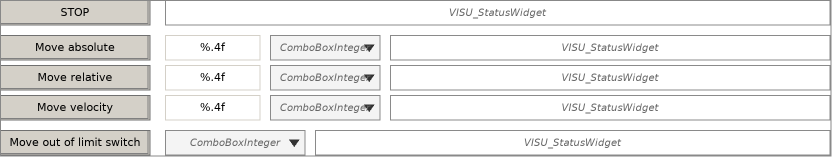
VISUALIZATION VISU_Axes_Commands_Movement  // 832x157
VAR_IN_OUT
    stop : AxesStopProcess;
    moveOutOfLimitSwitch : AxesMoveOutOfLimitSwitchProcess;
    moveAbsolute : AxesMoveAbsoluteProcess;
    moveRelative : AxesMoveRelativeProcess;
    moveVelocity : AxesMoveVelocityProcess;
    
    stopStatus : StatusWidget;
    moveOutOfLimitSwitchStatus : StatusWidget;
    moveAbsoluteStatus : StatusWidget;
    moveRelativeStatus : StatusWidget;
    moveVelocityStatus : StatusWidget;
END_VAR
    Button (0,0 150x25), "STOP", input disabled if: stop.statuses.enabledStatus.disabled
        OnMouseClick: execute { stop.request(); }
    Frame (165,0 665x25)
        shows VISU_StatusWidget(widget := stopStatus)
    Button (0,130 150x25), "Move out of limit switch", input disabled if: moveOutOfLimitSwitch.statuses.enabledStatus.disabled
        OnMouseClick: execute { moveOutOfLimitSwitch.do_request := TRUE; }
    Frame (315,130 515x25)
        shows VISU_StatusWidget(widget := moveOutOfLimitSwitchStatus)
    ComboBoxInteger (165,130 140x25), variable: moveOutOfLimitSwitch.set.switch, text list: 'LimitSwitchesTextList'
    Button (0,35 150x25), "Move absolute", input disabled if: moveAbsolute.statuses.enabledStatus.disabled
        OnMouseClick: execute { moveAbsolute.set.offset := 0.0; moveAbsolute.do_request := TRUE; }
    Textfield (165,35 95x25), "%.4f", text variable: moveAbsolute.set.value
        OnMouseClick: write the text variable via VisuDialogs.Numpad
    ComboBoxInteger (270,35 110x25), variable: moveAbsolute.set.units, text list: 'AxesMoveUnitsTextList'
    Frame (390,35 440x25)
        shows VISU_StatusWidget(widget := moveAbsoluteStatus)
    Button (0,65 150x25), "Move relative", input disabled if: moveRelative.statuses.enabledStatus.disabled
        OnMouseClick: execute { moveRelative.do_request := TRUE; }
    Textfield (165,65 95x25), "%.4f", text variable: moveRelative.set.value
        OnMouseClick: write the text variable via VisuDialogs.Numpad
    ComboBoxInteger (270,65 110x25), variable: moveAbsolute.set.units, text list: 'AxesMoveUnitsTextList'
    Frame (390,65 440x25)
        shows VISU_StatusWidget(widget := moveRelativeStatus)
    Button (0,95 150x25), "Move velocity", input disabled if: moveVelocity.statuses.enabledStatus.disabled
        OnMouseClick: execute { moveVelocity.do_request := TRUE; }
    Textfield (165,95 95x25), "%.4f", text variable: moveVelocity.set.value
        OnMouseClick: write the text variable via VisuDialogs.Numpad
    ComboBoxInteger (270,95 110x25), variable: moveVelocity.set.units, text list: 'AxesMoveVelocityUnitsTextList'
    Frame (390,95 440x25)
        shows VISU_StatusWidget(widget := moveVelocityStatus)
END_VISUALIZATION

(* stored: Version 1.1.0.1, ProductVersion 3.1.4019.2
   Visu VISU_Axes_Commands_Movement: Id {1887a7c8-2d38-4a4d-a0d0-85efb79e0b3f} *)
